FUNCTION_BLOCK Modbus
VAR_INPUT
END_VAR
VAR_OUTPUT
	ReadCount: LINT;
	ErrorCount: LINT;
END_VAR
VAR CONSTANT
	IO_COUNT: INT := 100;
END_VAR
VAR
	Self: REFERENCE TO Modbus;
	IO: ARRAY [0..IO_COUNT - 1] OF POINTER TO ModbusIo;
	IOIndex: INT;
	CurrentIoIndex: INT;
END_VAR

Self REF= THIS^;

METHOD AddIO : BOOL
VAR_INPUT
	Self: pointer TO ModbusIO {flag write};
END_VAR
IF IOIndex < IO_COUNT THEN
	IO[IOIndex] := Self;
	IOIndex := IOIndex + 1;
END_IF
END_METHOD

END_FUNCTION_BLOCK

(* stored: Version 1.1.0.1, ProductVersion 3.1.4024.3
   POU Modbus: Id {fd8b3be3-31b3-4684-971d-24fffd576038}, SpecialFunc None
   Method AddIO: Id {4be3b82a-4103-4e52-b617-e510c7e5594d} *)
